// TIA Portal V20 export
VAR_GLOBAL   // PLC tag table "Default tag table_1"
END_VAR
VAR_GLOBAL CONSTANT   // user constants
   "None(1)" : Pip := 65535;
   "Automatic update(1)" : Pip := 0;
   "PIP 1(1)" : Pip := 1;
   "PIP 2(1)" : Pip := 2;
   "PIP 3(1)" : Pip := 3;
   "PIP 4(1)" : Pip := 4;
   "PIP 5(1)" : Pip := 5;
   "PIP 6(1)" : Pip := 6;
   "PIP 7(1)" : Pip := 7;
   "PIP 8(1)" : Pip := 8;
   "PIP 9(1)" : Pip := 9;
   "PIP 10(1)" : Pip := 10;
   "PIP 11(1)" : Pip := 11;
   "PIP 12(1)" : Pip := 12;
   "PIP 13(1)" : Pip := 13;
   "PIP 14(1)" : Pip := 14;
   "PIP 15(1)" : Pip := 15;
   "PIP 16(1)" : Pip := 16;
   "PIP 17(1)" : Pip := 17;
   "PIP 18(1)" : Pip := 18;
   "PIP 19(1)" : Pip := 19;
   "PIP 20(1)" : Pip := 20;
   "PIP 21(1)" : Pip := 21;
   "PIP 22(1)" : Pip := 22;
   "PIP 23(1)" : Pip := 23;
   "PIP 24(1)" : Pip := 24;
   "PIP 25(1)" : Pip := 25;
   "PIP 26(1)" : Pip := 26;
   "PIP 27(1)" : Pip := 27;
   "PIP 28(1)" : Pip := 28;
   "PIP 29(1)" : Pip := 29;
   "PIP 30(1)" : Pip := 30;
   "PIP 31(1)" : Pip := 31;
   "PIP OB Servo(1)" : Pip := 32768;
   "Local~MC(1)" : Hw_SubModule := 51;
   "Local~Display(1)" : Hw_SubModule := 54;
   "Local~Exec(1)" : Hw_SubModule := 52;
   "Local(1)" : Hw_SubModule := 49;
   "Local~PROFINET_interface_1(1)" : Hw_Interface := 64;
   "Local~PROFINET_interface_1~Port_1(1)" : Hw_Interface := 65;
   "Local~PROFINET_interface_1~Port_2(1)" : Hw_Interface := 66;
   "Local~PROFINET_interface_2(1)" : Hw_Interface := 72;
   "Local~PROFINET_interface_2~Port_1(1)" : Hw_Interface := 73;
   "Local~Virtual_communication_interface(1)" : Hw_Interface := 135;
   "Local~License_Manager(1)" : Hw_SubModule := 42;
   "Local~PROFINET_IO-System(1)" : Hw_IoSystem := 257;
   "IOLink_21~Proxy(1)" : Hw_SubModule := 258;
   "IOLink_21~IODevice(1)" : Hw_Device := 273;
   "IOLink_21~PN-IO(1)" : Hw_Interface := 259;
   "IOLink_21~PN-IO~Port_X01_10_100_MBit_s(1)" : Hw_Interface := 260;
   "IOLink_21~PN-IO~Port_X02_10_100_MBit_s(1)" : Hw_Interface := 261;
   "IOLink_21~Head(1)" : Hw_SubModule := 262;
   "Digital_In_(A)_Dig__(B)_1(1)" : Hw_SubModule := 266;
   "IOLink_21~LMD01(1)" : Hw_SubModule := 263;
   "IOLink_21~LMD01~Status_Control_Module(1)" : Hw_SubModule := 264;
   "IOLink_21~LMD01~XAC(1)" : Hw_SubModule := 322;
   "IOLink_22~Proxy(1)" : Hw_SubModule := 311;
   "IOLink_22~IODevice(1)" : Hw_Device := 309;
   "IOLink_22~PN-IO(1)" : Hw_Interface := 312;
   "IOLink_22~PN-IO~Port_X01_10_100_MBit_s(1)" : Hw_Interface := 313;
   "IOLink_22~PN-IO~Port_X02_10_100_MBit_s(1)" : Hw_Interface := 314;
   "IOLink_22~Head(1)" : Hw_SubModule := 315;
   "IOLink_22~LMD02(1)" : Hw_SubModule := 316;
   "IOLink_22~LMD02~Status_Control_Module(1)" : Hw_SubModule := 317;
   "GR2_SEW-EURODRIVE-UHX45~Proxy(1)" : Hw_SubModule := 340;
   "GR2_SEW-EURODRIVE-UHX45~IODevice(1)" : Hw_Device := 338;
   "GR2_SEW-EURODRIVE-UHX45~PN-IO(1)" : Hw_Interface := 341;
   "GR2_SEW-EURODRIVE-UHX45~PN-IO~Port_1_-_RJ45_(X40)(1)" : Hw_Interface := 342;
   "GR2_SEW-EURODRIVE-UHX45~PN-IO~Port_2_-_RJ45_(X41)(1)" : Hw_Interface := 343;
   "GR2_SEW-EURODRIVE-UHX45~Head(1)" : Hw_SubModule := 344;
   "GR2_SEW-EURODRIVE-UHX45~Module_I_O_(64_words)_1(1)" : Hw_SubModule := 353;
   "GR2_SEW-EURODRIVE-UHX45~Empty_8(1)" : Hw_SubModule := 352;
   "GR2_SEW-EURODRIVE-UHX45~Empty_7(1)" : Hw_SubModule := 351;
   "GR2_SEW-EURODRIVE-UHX45~Empty_6(1)" : Hw_SubModule := 350;
   "GR2_SEW-EURODRIVE-UHX45~Empty_5(1)" : Hw_SubModule := 349;
   "GR2_SEW-EURODRIVE-UHX45~Empty_4(1)" : Hw_SubModule := 348;
   "GR2_SEW-EURODRIVE-UHX45~Empty_3(1)" : Hw_SubModule := 347;
   "GR2_SEW-EURODRIVE-UHX45~Empty_2(1)" : Hw_SubModule := 346;
   "GR2_SEW-EURODRIVE-UHX45~Empty_1(1)" : Hw_SubModule := 345;
   "OB_Task_1ms(1)" : OB_Cyclic := 31;
   "OB_Task_100ms(1)" : OB_Cyclic := 32;
   "OB_Task_Comm(1)" : OB_Cyclic := 38;
   "OB_ProgrammingError(1)" : OB_Any := 121;
   "SensorCheck_FallingEdge(1)" : USInt := 0;
   "SensorCheck_Off(1)" : USInt := 3;
   "SensorCheck_On(1)" : USInt := 2;
   "SensorCheck_RisingEdge(1)" : USInt := 1;
   "GR_RIO_20~Head(1)" : Hw_SubModule := 329;
   "GR_RIO_20~PROFINET_interface(1)" : Hw_Interface := 330;
   "GR_RIO_20~PROFINET_interface~Port_1(1)" : Hw_Interface := 331;
   "GR_RIO_20~PROFINET_interface~Port_2(1)" : Hw_Interface := 332;
   "GR_RIO_20~DI_16x24VDC_ST_1(1)" : Hw_SubModule := 333;
   "GR_RIO_20~DI_16x24VDC_ST_2(1)" : Hw_SubModule := 334;
   "GR_RIO_20~DI_16x24VDC_ST_3(1)" : Hw_SubModule := 335;
   "GR_RIO_20~DQ_16x24VDC_0_5A_ST_1(1)" : Hw_SubModule := 336;
   "GR_RIO_20~DQ_16x24VDC_0_5A_ST_2(1)" : Hw_SubModule := 337;
   "GR_RIO_20~Proxy(1)" : Hw_SubModule := 328;
   "GR_RIO_20~IODevice(1)" : Hw_Device := 326;
   "GR_RIO_20~Server_module_1(1)" : Hw_SubModule := 354;
   "IOLink_21~LMD01~X1RD1(1)" : Hw_SubModule := 265;
   "IOLink_21~LMD01~X2RD1(1)" : Hw_SubModule := 267;
   "OB_Task_Startup(1)" : OB_STARTUP := 100;
   "IDLE(1)" : UInt := 0;
   "JOG_POS(1)" : UInt := 100;
   "JOG_SPD(1)" : UInt := 101;
   "SPD_CTRL(1)" : UInt := 200;
   "HOMING(1)" : UInt := 300;
   "HOMEING_OFFSET(1)" : UInt := 301;
   "ABS_POS(1)" : UInt := 400;
   "REL_POS(1)" : UInt := 401;
   "BRK_OPEN(1)" : UInt := 700;
   "OB_Task_10ms(1)" : OB_Cyclic := 30;
   "OB_Task_Aperiodic(1)" : OB_PCYCLE := 1;
   "OB_Task_10ms_Test(1)" : OB_Cyclic := 33;
   "TB5000_Offset(1)" : UInt := 41;
   "Local~Common(1)" : Hw_SubModule := 50;
   "Local~Device(1)" : Hw_Device := 32;
   "Local~Configuration(1)" : Hw_SubModule := 33;
   "IOLink_22~LMD02~FLD(1)" : Hw_SubModule := 281;
   "IOLink_22~LMD02~GDL(1)" : Hw_SubModule := 282;
   "IOLink_22~LMD02~GDF(1)" : Hw_SubModule := 283;
   "IOLink_22~LMD02~GDR(1)" : Hw_SubModule := 284;
   "IOLink_22~LMD02~Inactive_(A_B)(1)" : Hw_SubModule := 269;
   "IOLink_22~LMD02~Inactive_(A_B)_1(1)" : Hw_SubModule := 275;
   "IOLink_22~LMD02~Inactive_(A_B)_2(1)" : Hw_SubModule := 276;
   "IOLink_22~LMD02~Inactive_(A_B)_3(1)" : Hw_SubModule := 277;
   "IOLink_21~LMD01~Inactive_(A_B)(1)" : Hw_SubModule := 268;
   "IOLink_21~LMD01~Inactive_(A_B)_1(1)" : Hw_SubModule := 270;
   "IOLink_21~LMD01~Inactive_(A_B)_2(1)" : Hw_SubModule := 271;
   "IOLink_21~LMD01~Inactive_(A_B)_3(1)" : Hw_SubModule := 272;
END_VAR
